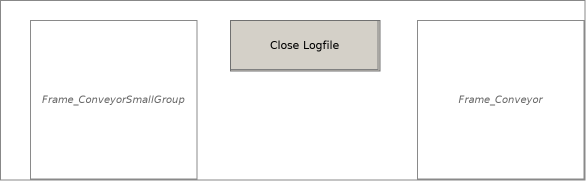
VISUALIZATION VISU_MEDIATOR_TEST  // 586x181
    Frame (30,20 167x159)
        shows Frame_ConveyorSmallGroup(vio_fbConveyor1 := MEDIATOR_TEST.aConveyorPeers[1], vio_fbConveyor2 := MEDIATOR_TEST.aConveyorPeers[2], vio_fbConveyor3 := MEDIATOR_TEST.aConveyorPeers[3], vio_fbConveyor4 := MEDIATOR_TEST.aConveyorPeers[4])
    Button (230,20 150x51), "Close Logfile"
        tap MEDIATOR_TEST.bCloseFile
    Frame (417,20 167x159)
        shows Frame_Conveyor(vio_fbConveyor := MEDIATOR_TEST.aConveyorPeers[1])
END_VISUALIZATION

(* stored: Version 1.1.0.1, ProductVersion 3.1.4022.16
   Visu VISU_MEDIATOR_TEST: Id {45df7361-aa3c-4eca-88d0-52b567287016} *)
